FUNCTION_BLOCK FB_LensMock EXTENDS FB_FalliblePublicMock IMPLEMENTS I_Lens
VAR
    sMaterialName : T_MaxString;
    nMultiplier : INT;
    fbRadius : FB_QuantityLREALPublic(Units := 'm');
END_VAR


METHOD GetRadius
VAR_OUTPUT
    Radius : FB_QuantityLREALPublic(Units := '');
END_VAR

Radius := fbRadius;
END_METHOD


PROPERTY MaterialFormula : T_MaxString
GET

MaterialFormula := sMaterialName;
END_GET
SET

sMaterialName := MaterialFormula;
END_SET
END_PROPERTY


PROPERTY Multiplier : INT
GET

Multiplier := nMultiplier;
END_GET
SET

nMultiplier := Multiplier;
END_SET
END_PROPERTY


METHOD SetRadius
VAR_INPUT
    Radius : I_QuantityLREAL;
END_VAR

fbRadius.Copy(QuantityToCopy := Radius);
END_METHOD


METHOD SetValid
VAR
    nIndex : INT;
END_VAR

ClearError();
sMaterialName := 'Be';
nMultiplier := 1;
fbRadius.Val := 1.0;
fbRadius.Units := 'm';
fbRadius.ClearError();
END_METHOD

END_FUNCTION_BLOCK

(* stored: Version 1.1.0.1
   POU FB_LensMock: Id {8e5e1b9f-38a8-4173-b9ab-660968f25168}, SpecialFunc None
   Method GetRadius: Id {1e936b74-6ae1-48de-8fb7-a0e4f6da68ed}
   Property MaterialFormula: Id {d5018cf9-ae4a-4b2b-bb13-fbe3f764b9b8}
   Get Get: Id {8f4c5ef5-2e6e-4653-bf7c-5b3586634ae6}
   Set Set: Id {68152525-8594-40ce-9e2d-cd99711db00a}
   Property Multiplier: Id {61aeae02-dce5-4640-a899-9989b314e3b7}
   Get Get: Id {3c7cbc25-d2b2-4f4a-8456-b8ec28707001}
   Set Set: Id {520f5cdf-d172-4950-99f3-6e7264aedd43}
   Method SetRadius: Id {fc452968-65ff-4321-92f9-1af7b8d51ad8}
   Method SetValid: Id {a370019b-6194-4481-bd92-0da263acb531} *)
